// TwinCAT 3 PLC project supervisor
// ProgramVersion: 3.1.4023.0
// libraries:
//   Tc2_DataExchange, * (Beckhoff Automation GmbH)
//   Tc2_Standard, * (Beckhoff Automation GmbH)
//   Tc2_System, * (Beckhoff Automation GmbH)
//   Tc3_Module, * (Beckhoff Automation GmbH)
// project tree:
//   GVLs/ GVL.TcGVL
//   / PlcTask.TcTTO
//   POUs/ MAIN.TcPOU, POU_copyXmeasXmv.TcPOU
// real-time tasks:
//   TASK PlcTask: cycle T#10ms, priority 20, ADS port 350

CONFIGURATION supervisor
    RESOURCE PLC ON TwinCAT3
        TASK PlcTask(INTERVAL := T#10ms, PRIORITY := 20);
        PROGRAM MAIN WITH PlcTask : MAIN;
    END_RESOURCE
END_CONFIGURATION

// ---- GVLs/GVL.TcGVL
{attribute 'qualified_only'}
VAR_GLOBAL
	// setpoints
	PROD_RATE_SP					:	LREAL	:= 22.89;	// production rate
	L_STRIPPER_SP					:	LREAL	:= 50.0;	// stripper level
	L_SEPARATOR_SP					:	LREAL	:= 50.0;	// separator level
	L_REACTOR_SP					:	LREAL	:= 65.0;	// reactor level
	P_REACTOR_SP					:	LREAL	:= 2800;	// reactor pressure
	PCT_G_SP						:	LREAL	:= 53.8;	// Mole percent G
	YA_SP							: 	LREAL	:= (100.0*32.2/(32.2+18.8));	// yA 
	YAC_SP							:	LREAL	:= 32.2+18.8;	// yAC
	T_REACTOR_SP					:	LREAL	:= 122.9;	// reactor temperature
	RECYC_VALVE_SP					:	LREAL	:= 0.0;		// Recycle valve position
	STEAM_VALVE_SP					:	LREAL	:= 0.0;		// Steam valve position
	L_AGITATOR_SP					:	LREAL	:= 100.0;	// agitator setting		
	
	// Intermediate values
	Fp							:	LREAL; // production rate used by reactor, stripper, and separator
	SepTempSP					:	LREAL; // tmp sp used by separator
	RI							:	ARRAY[1..7] OF LREAL;	// ratio trimming outputs
	EADJ						:	LREAL;	// adjustment to production rate

	// actual production metrics
	COST						:	LREAL :=0.0;
	PctG						:	LREAL :=0.0;

	// process variables
	XMEAS						:	ARRAY[1..41] OF LREAL;  // this is formed from the variable copied from the various process control parts
	XMEAS_FROM_REACTOR			:	ARRAY[1..16] OF LREAL;
	XMEAS_FROM_SEPARATOR		:	ARRAY[1..15] OF LREAL;
	XMEAS_FROM_STRIPPER			:	ARRAY[1..10] OF LREAL;
	
	XMV							:	ARRAY[1..12] OF LREAL;  // this is formed from the variable copied from the various process control parts
	XMV_FROM_REACTOR			:	ARRAY[1..7] OF LREAL;
	XMV_FROM_SEPARATOR			:	ARRAY[1..3] OF LREAL;
	XMV_FROM_STRIPPER			:	ARRAY[1..2] OF LREAL;
	
	// shutdown indicator
	SD_FLAG						: 	BOOL	:= FALSE;
	
	// Disturbance vector
	IDV							:	ARRAY[1..20] OF LREAL	:= [0,0,0,0,0,0,0,0,0,0,0,0];

END_VAR

// ---- POUs/MAIN.TcPOU
PROGRAM MAIN
VAR
	
	tonCopy :	TON;
	checkPctG: LREAL;
END_VAR


tonCopy(in:=NOT(tonCopy.Q), PT:=T#900MS);

IF tonCopy.Q THEN
	POU_copyXmeasXmv();
END_IF

END_PROGRAM

// ---- POUs/POU_copyXmeasXmv.TcPOU
PROGRAM POU_copyXmeasXmv
VAR
	II: INT := 1;
	
	iiXmeasReactor			:	ARRAY[1..16] OF INT := [1,2,3,4,5,6,7,8,9,21,23,24,25,26,27,28];
	iiXmvReactor			:	ARRAY[1..7] OF INT := [1,2,3,4,10,11,12];
	
	iiXmeasSep				:	ARRAY[1..15] OF INT := [10,11,12,13,14,20,22,29,30,31,32,33,34,35,36];
	iiXmvSep				:	ARRAY[1..3] OF INT := [5,6,7];
	
	iiXmeasStrip			:	ARRAY[1..10] OF INT := [15,16,17,18,19,37,38,39,40,41];
	iiXmvStrip				:	ARRAY[1..2] OF INT := [8, 9];	
END_VAR



// XMEAS from REACTOR
FOR II := 1 TO SIZEOF(iiXmeasReactor)/SIZEOF(iiXmeasReactor[1]) DO
	GVL.XMEAS[iiXmeasReactor[ii]]:=GVL.XMEAS_FROM_REACTOR[II];
END_FOR

// XMV FROMfrom REACTOR
FOR II := 1 TO SIZEOF(iiXmvReactor)/SIZEOF(iiXmvReactor[1]) DO
	GVL.XMV[iiXmvReactor[ii]]:=GVL.XMV_FROM_REACTOR[II];
END_FOR

// XMEAS from SEPARATOR
FOR II := 1 TO SIZEOF(iiXmeasSep)/SIZEOF(iiXmeasSep[1]) DO
	GVL.XMEAS[iiXmeasSep[ii]]:=GVL.XMEAS_FROM_SEPARATOR[II];
END_FOR

// XMV FROMfrom SEPARATOR
FOR II := 1 TO SIZEOF(iiXmvSep)/SIZEOF(iiXmvSep[1]) DO
	GVL.XMV[iiXmvSep[ii]]:=GVL.XMEAS_FROM_SEPARATOR[II];
END_FOR

// XMEAS from STRIPPER
FOR II := 1 TO SIZEOF(iiXmeasStrip)/SIZEOF(iiXmeasStrip[1]) DO
	GVL.XMEAS[iiXmeasStrip[ii]]:=GVL.XMEAS_FROM_STRIPPER[II];
END_FOR

// XMV FROMfrom STRIPPER
FOR II := 1 TO SIZEOF(iiXmvStrip)/SIZEOF(iiXmvStrip[1]) DO
	GVL.XMV[iiXmvStrip[ii]]:=GVL.XMEAS_FROM_STRIPPER[II];
END_FOR

END_PROGRAM
